# EPICS substitutions: iocBoot/ioc13Linux/BNC_505.substitutions
# This loads the records that apply to the entire BNC-505.
file "$(DELAYGEN)/delaygenApp/Db/BNC_505.db"
{
pattern
{P,            R,         PORT    }
{13Linux:,     BNC1:,     serial1 }
}

# This loads the records for each BNC-505 output.
file "$(DELAYGEN)/delaygenApp/Db/BNC_505_Pn.db"
{
pattern
{P,            R,        PORT,      N}
{13Linux:,     BNC1:,    serial1,   1}
{13Linux:,     BNC1:,    serial1,   2}
}
